FUNCTION Convert_UDINT_TO_STRING : Hresult
VAR_INPUT
	in : UDINT;
	out : REFERENCE TO STRING;
END_VAR
VAR
	converted : STRING;
END_VAR
VAR CONSTANT
	INCOMPATIBLE : HRESULT := 16#9811070E;
END_VAR

converted := UDINT_TO_STRING(in);

IF (STRING_TO_UDINT(converted) <> in) THEN
	Convert_UDINT_TO_STRING := INCOMPATIBLE;
	RETURN;
END_IF

out := converted;

END_FUNCTION

(* stored: Version 1.1.0.1, ProductVersion 3.1.4024.12
   POU Convert_UDINT_TO_STRING: Id {14bb7a3a-4d0e-4113-9060-5aca22f53a69}, SpecialFunc None *)
